// Mitsubishi GX Works2 project: 1   PLC: FX3U/FX3UC

TYPE struct : STRUCT
END_STRUCT END_TYPE

// global labels: Global1
VAR_GLOBAL
  测试_4 : 测试;
END_VAR

PROGRAM MAIN
VAR
  测试_1 : 测试;
  测试_2 : 测试;
  测试_3 : 测试;
  测试_5 : 测试;
  测试_8 : 测试;
  测试_9 : 测试;
END_VAR
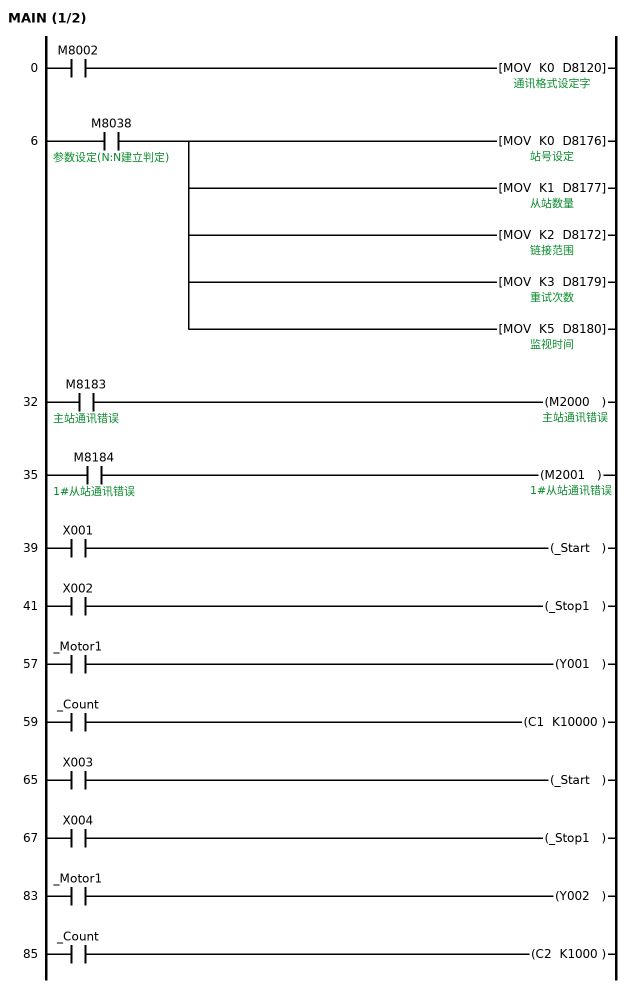
0     LD      M8002
      MOV     K0 D8120  ; 通讯格式设定字
6     LD      M8038  ; 参数设定(N:N建立判定)
      MOV     K0 D8176  ; 站号设定
      MOV     K1 D8177  ; 从站数量
      MOV     K2 D8172  ; 链接范围
      MOV     K3 D8179  ; 重试次数
      MOV     K5 D8180  ; 监视时间
32    LD      M8183  ; 主站通讯错误
      OUT     M2000  ; 主站通讯错误
35    LD      M8184  ; 1#从站通讯错误
      OUT     M2001  ; 1#从站通讯错误
; FB BLK START 测试(测试_1)
39    LD      X001
      OUT     _Start
41    LD      X002
      OUT     _Stop1
; FB START
; FB_NAME 测试
; INSTANCE_NAME 测试_1
; FB IN_B:Start
; FB OUT_Motor1:B
; FB IN_B:Stop1
; FB OUT_Count:B
; FB IN_B:ST1
; FB OUT_I_O:W
; FB IN_B:ST2
; FB IN_B:ST3
; FB IN_B:ST4
; FB IN_W:I_O
; FB END
57    LD      _Motor1
      OUT     Y001
59    LD      _Count
      OUT     C1 K10000
; FB BLK END
; FB BLK START 测试(测试_2)
65    LD      X003
      OUT     _Start
67    LD      X004
      OUT     _Stop1
; FB START
; FB_NAME 测试
; INSTANCE_NAME 测试_2
; FB IN_B:Start
; FB OUT_Motor1:B
; FB IN_B:Stop1
; FB OUT_Count:B
; FB IN_B:ST1
; FB OUT_I_O:W
; FB IN_B:ST2
; FB IN_B:ST3
; FB IN_B:ST4
; FB IN_W:I_O
; FB END
83    LD      _Motor1
      OUT     Y002
85    LD      _Count
      OUT     C2 K1000
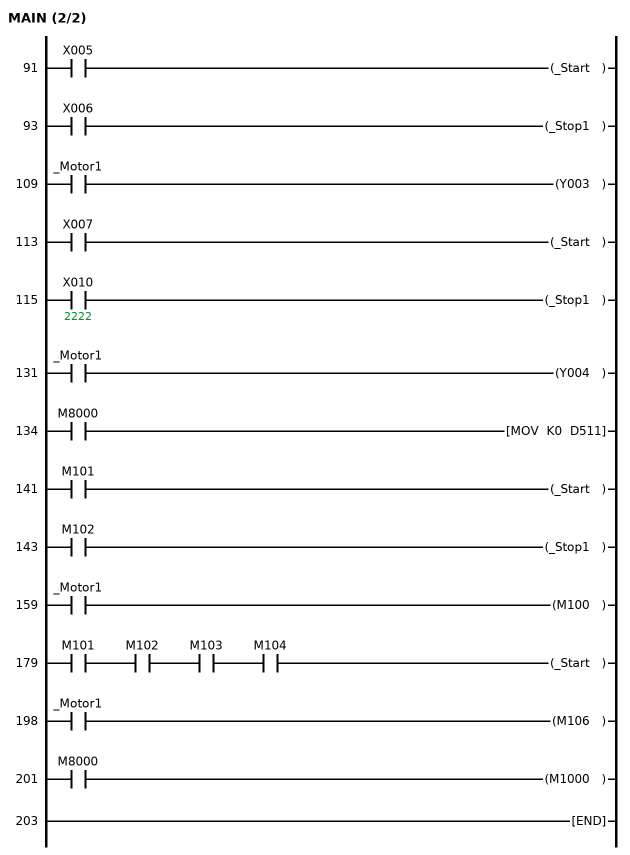
; FB BLK END
; FB BLK START 测试(测试_3)
91    LD      X005
      OUT     _Start
93    LD      X006
      OUT     _Stop1
; FB START
; FB_NAME 测试
; INSTANCE_NAME 测试_3
; FB IN_B:Start
; FB OUT_Motor1:B
; FB IN_B:Stop1
; FB OUT_Count:B
; FB IN_B:ST1
; FB OUT_I_O:W
; FB IN_B:ST2
; FB IN_B:ST3
; FB IN_B:ST4
; FB IN_W:I_O
; FB END
109   LD      _Motor1
      OUT     Y003
; FB BLK END
; FB BLK START 测试(测试_4)
113   LD      X007
      OUT     _Start
115   LD      X010  ; 2222
      OUT     _Stop1
; FB START
; FB_NAME 测试
; INSTANCE_NAME 测试_4
; FB IN_B:Start
; FB OUT_Motor1:B
; FB IN_B:Stop1
; FB OUT_Count:B
; FB IN_B:ST1
; FB OUT_I_O:W
; FB IN_B:ST2
; FB IN_B:ST3
; FB IN_B:ST4
; FB IN_W:I_O
; FB END
131   LD      _Motor1
      OUT     Y004
; FB BLK END
134   LD      M8000
      MOV     K0 D511
; FB BLK START 测试(测试_5)
141   LD      M101
      OUT     _Start
143   LD      M102
      OUT     _Stop1
; FB START
; FB_NAME 测试
; INSTANCE_NAME 测试_5
; FB IN_B:Start
; FB OUT_Motor1:B
; FB IN_B:Stop1
; FB OUT_Count:B
; FB IN_B:ST1
; FB OUT_I_O:W
; FB IN_B:ST2
; FB IN_B:ST3
; FB IN_B:ST4
; FB IN_W:I_O
; FB END
159   LD      _Motor1
      OUT     M100
; FB BLK END
; FB BLK START 测试(测试_8)
; FB START
; FB_NAME 测试
; INSTANCE_NAME 测试_8
; FB IN_B:Start
; FB OUT_Motor1:B
; FB IN_B:Stop1
; FB OUT_Count:B
; FB IN_B:ST1
; FB OUT_I_O:W
; FB IN_B:ST2
; FB IN_B:ST3
; FB IN_B:ST4
; FB IN_W:I_O
; FB END
; FB BLK END
; FB BLK START 测试(测试_9)
179   LD      M101
      AND     M102
      AND     M103
      AND     M104
      OUT     _Start
; FB START
; FB_NAME 测试
; INSTANCE_NAME 测试_9
; FB IN_B:Start
; FB OUT_Motor1:B
; FB IN_B:Stop1
; FB OUT_Count:B
; FB IN_B:ST1
; FB OUT_I_O:W
; FB IN_B:ST2
; FB IN_B:ST3
; FB IN_B:ST4
; FB IN_W:I_O
; FB END
198   LD      _Motor1
      OUT     M106
; FB BLK END
201   LD      M8000
      OUT     M1000
203   END
END_PROGRAM

FUNCTION_BLOCK 测试
VAR_INPUT
  Start : BOOL;  (* 启动按钮 *)
  Stop1 : BOOL;  (* 停止按钮 *)
END_VAR
VAR_OUTPUT
  Motor1 : BOOL;  (* 电机 *)
END_VAR
VAR
  array_1 : ARRAY [1..3] OF BOOL;  (* 数组 *)
  hello : BOOL;  (* 你好 *)
  worild : BOOL;
  辅助位 : BOOL;
  w1 : BOOL;
END_VAR
VAR_INPUT
  ST1 : BOOL;
  ST2 : BOOL;
  ST3 : BOOL;
  ST4 : BOOL;
END_VAR
VAR_OUTPUT
  Count : BOOL;  (* 计数 *)
END_VAR
VAR
  hh : BOOL;
  hou : BOOL;
END_VAR
VAR_IN_OUT
  I_O : INT;
END_VAR
VAR
  fb1_1 : fb1;
END_VAR
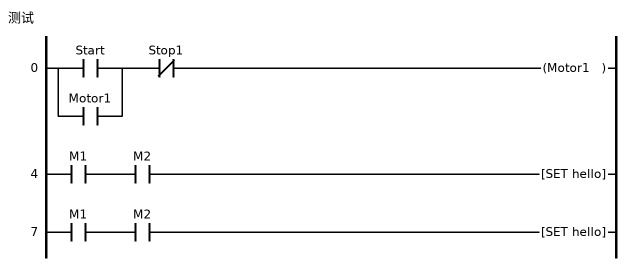
0     LD      Start
      OR      Motor1
      ANI     Stop1
      OUT     Motor1
4     LD      M1
      AND     M2
      SET     hello
7     LD      M1
      AND     M2
      SET     hello
; FB BLK START fb1(fb1_1)
; FB START
; FB_NAME fb1
; INSTANCE_NAME fb1_1
; FB IN_B:heh1
; FB OUT_heh2:B
; FB END
; FB BLK END
END_FUNCTION_BLOCK

FUNCTION_BLOCK fb1
VAR_INPUT
  heh1 : BOOL;
END_VAR
VAR_OUTPUT
  heh2 : BOOL;
END_VAR
END_FUNCTION_BLOCK

PROGRAM MAIN1
VAR
  asd : 123;
  主控启动 : BOOL;
  扫模完成 : BOOL;
END_VAR
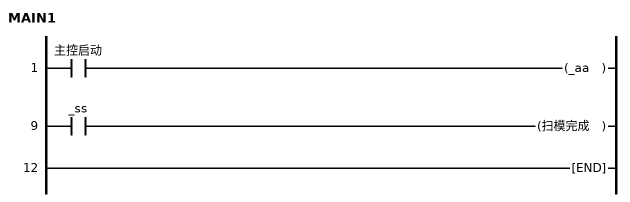
; FB BLK START 123(asd)
1     LD      主控启动
      OUT     _aa
; FB START
; FB_NAME 123
; INSTANCE_NAME asd
; FB IN_B:aa
; FB OUT_ss:B
; FB END
9     LD      _ss
      OUT     扫模完成
; FB BLK END
12    END
END_PROGRAM

FUNCTION_BLOCK 123
VAR_INPUT
  aa : BOOL;
END_VAR
VAR
  程序启动 : BOOL;
END_VAR
VAR_OUTPUT
  ss : BOOL;
END_VAR
VAR
  SS1 : BOOL;
  SS2 : BOOL;
  SS3 : BOOL;
  SS4 : BOOL;
  SS5 : BOOL;
  SS6 : BOOL;
  SS7 : BOOL;
  SS8 : BOOL;
  SS9 : BOOL;
  SS10 : BOOL;
  SS11 : BOOL;
  SS12 : BOOL;
  SS13 : BOOL;
  SS14 : BOOL;
  SS15 : BOOL;
  SS16 : BOOL;
  SS17 : BOOL;
  SS18 : BOOL;
  SS19 : BOOL;
  SS20 : BOOL;
  SS21 : BOOL;
  SS22 : BOOL;
  SS23 : BOOL;
  SS24 : BOOL;
  SS25 : BOOL;
  SS26 : BOOL;
  SS27 : BOOL;
  SS28 : BOOL;
  SS29 : BOOL;
  SS30 : BOOL;
  SS31 : BOOL;
  SS32 : BOOL;
  SS33 : BOOL;
  SS34 : BOOL;
  SS35 : BOOL;
  SS36 : BOOL;
  SS37 : BOOL;
  SS38 : BOOL;
  SS39 : BOOL;
  SS40 : BOOL;
  SS41 : BOOL;
  SS42 : BOOL;
  SS43 : BOOL;
  SS44 : BOOL;
  SS45 : BOOL;
  SS46 : BOOL;
  SS47 : BOOL;
  SS48 : BOOL;
  SS49 : BOOL;
  SS50 : BOOL;
  SS51 : BOOL;
  SS52 : BOOL;
  SS53 : BOOL;
  SS54 : BOOL;
  SS55 : BOOL;
  SS56 : BOOL;
  SS57 : BOOL;
  SS68 : BOOL;
  SS69 : BOOL;
  SS70 : BOOL;
  SS71 : BOOL;
  SS72 : BOOL;
  SS73 : BOOL;
  SS74 : BOOL;
  SS75 : BOOL;
  SS76 : BOOL;
  SS77 : BOOL;
  SS58 : BOOL;
  SS59 : BOOL;
  SS60 : BOOL;
  SS61 : BOOL;
  SS62 : BOOL;
  SS63 : BOOL;
  SS64 : BOOL;
  SS65 : BOOL;
  SS66 : BOOL;
  SS67 : BOOL;
  SS78 : BOOL;
  SS79 : BOOL;
  SS80 : BOOL;
  SS81 : BOOL;
  SS82 : BOOL;
  SS83 : BOOL;
  SS84 : BOOL;
  SS85 : BOOL;
  SS86 : BOOL;
  SS87 : BOOL;
  SS88 : BOOL;
  SS89 : BOOL;
  SS90 : BOOL;
  SS91 : BOOL;
  SS92 : BOOL;
  SS93 : BOOL;
  SS94 : BOOL;
  SS95 : BOOL;
  SS96 : BOOL;
  SS97 : BOOL;
  SS98 : BOOL;
  SS99 : BOOL;
  SS100 : BOOL;
  SS101 : BOOL;
  SS102 : BOOL;
  SS103 : BOOL;
  SS104 : BOOL;
  SS105 : BOOL;
  SS106 : BOOL;
  SS107 : BOOL;
END_VAR
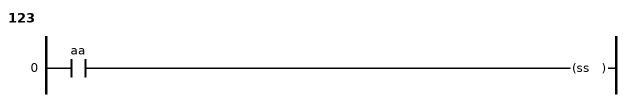
0     LD      aa
      OUT     ss
END_FUNCTION_BLOCK
